// SIMATIC STEP 7 (V5.x) project Station4
// CPU: CPU 314C-2 PN/DP

SYMBOL_TABLE
"CYC_INT5"	OB 35	OB 35	// Cyclic Interrupt 5
END_SYMBOL_TABLE
